Yaskawa INFORM job: FILLET_WELD.JBI

/JOB
//NAME FILLET_WELD
//POS
///NPOS 8,0,0,0,0,0
///TOOL 5
///POSTYPE PULSE
///PULSE
C00000=-4,-50478,-58434,17,-74948,475
C00001=1480,76606,32326,19738,-111363,-60504
C00002=1480,78430,31592,19470,-109599,-60831
C00003=-5354,79690,39005,7029,-114495,-68028
C00004=-5264,81068,38517,6822,-113056,-68133
C00005=3196,80598,37559,1297,-113107,-70556
C00006=3494,78071,38605,1199,-115808,-70622
C00007=-4,-50479,-58434,19,-74959,471
//INST
///DATE 2024/07/11 16:39
///ATTR SC,RW
///GROUP1 RB1
NOP
MOVJ C00000 VJ=4.00
COMM MOVJ C00001 VJ=4.00
COMM MOVL C00002 V=11.0
MOVJ C00003 VJ=4.00
MOVL C00004 V=11.0
DOUT OT#(17) ON
ARCON AC=60 AVP=80
COMM DOUT OT#(17) OFF
MOVL C00005 V=1.5
DOUT OT#(17) OFF
COMM TIMER T=1.00
ARCOF
MOVL C00006 V=11.0
MOVJ C00007 VJ=4.00
END
